// TIA Portal V19 export
TYPE "LEXCHANGETRAY_typeConstraintRollerEm_signalTM_Monitor"
// stored: Access Published
   STRUCT
      detectionBeforePalletPositioning : Bool;   // 托盘定位前检测
      positioningPinCylinderHomePositionDetection2 : Bool;   // 定位销气缸原位检测2
      cellLiftingCylinderHomePositionDetection2 : Bool;   // 电池顶升气缸原位检测2
      positioningPinCylinderWorkingPositionDetection2 : Bool;   // 定位销气缸工作位检测2
      trayLiftingCylinderWorkingPositionDetection : Bool;   // 托盘顶升气缸工作位检测
      cellLiftingCylinderWorkingPositionDetection2 : Bool;   // 电池顶升气缸工作位检测2
      cellLiftingCylinderHomePositionDetection1 : Bool;   // 电池顶升气缸原位检测1
      trayEntryDetection : Bool;   // 托盘进入检测
      trayLiftingCylinderHomePositionDetection : Bool;   // 托盘顶升气缸原位检测
      positiveLimitForCellJackingAndTransplanting : Bool;   // 电池顶升移栽正限
      negativeLimitForCellJackingAndTransplanting : Bool;   // 电池顶升移栽负限
      cellLiftingCylinderWorkingPositionDetection1 : Bool;   // 电池顶升气缸工作位检测1
      positioningPinCylinderHomePositionDetection1 : Bool;   // 定位销气缸原位检测1
      positioningPinCylinderWorkingPositionDetection1 : Bool;   // 定位销气缸工作位检测1
      trayInPlaceDetection : Bool;   // 托盘到位检测
      originalForCellJackingAndTransplanting : Bool;   // 电池顶升移栽原点
      palletScrewAntiReverseDetection : Bool;   // 托盘螺杆防反检测
      detectionAfterTrayPositioning : Bool;   // 托盘定位后检测
      trayLiftingCylinderHomePositionDetection1 : Bool;
      trayLiftingCylinderWorkingPositionDetection1 : Bool;
      simulationed : Bool;
   END_STRUCT;
END_TYPE
